(* PLC project Sem nome, Desconhecido Sem nome 1 *)
(* stored: creationDateTime 2023-06-19T15:21:12, modificationDateTime 2023-06-19T15:21:12 *)

CONFIGURATION Config0
  RESOURCE Res0 ON PLC
  END_RESOURCE
END_CONFIGURATION
